PROGRAM Torque_Scaling
VAR
	Rotor_Actual_Torque_Scaled : REAL;
END_VAR

Rotor_Actual_Torque_Scaled := INT_TO_REAL(GVL_Pelletizer.MyPelletizer.Rotor_VFD.VFD_Actual_Torque) / 10;

END_PROGRAM

(* stored: Version 1.1.0.1, ProductVersion 3.1.4024.12
   POU Torque_Scaling: Id {8e970592-64c0-43ad-8110-566d9f1a776b}, SpecialFunc None *)
